Yaskawa INFORM job: ROVI_RECIPE.JBI

/JOB
//NAME ROVI_RECIPE
///FOLDERNAME ROVI
//POS
///NPOS 0,0,0,0,0,0
//ARGINFO
///ARGTYPE I,,,,,,,
///COMMENT
RECIPE_NAME







//INST
///DATE 2019/12/05 17:26
///ATTR SC,RW
///GROUP1 RB1
///LVARS 1,3,0,0,0,0,0,0
NOP
GETARG LI002 IARG#(1)
SET LI000 I092
SET LI001 0
*RECIPE
SET I080 LI002
SET B080 3
WAIT B080=255
INC LI001
IFTHENEXP I080<>0
	 RET I080 IF LI001>=LI000
	 TIMER T=0.500
	 JUMP *RECIPE
ENDIF
RET I080
END
